PROGRAM MAIN
VAR
    rTrig : R_TRIG;
END_VAR

rTrig(CLK := GVL.BoutonSelecteur);

GVL.LumiereDroite := FALSE;
GVL.LumiereGauche := FALSE;

IF GVL.BoutonVirtuel THEN
    IF GVL.BoutonSelecteur THEN
        GVL.LumiereDroite := TRUE;
    ELSE
        GVL.LumiereGauche := TRUE;
    END_IF
END_IF;

IF rTrig.Q AND GVL.BoutonVirtuel THEN
    IF GVL.BoutonSelecteur THEN
        GVL.CounterLumiereDroiteAllumer := GVL.CounterLumiereDroiteAllumer + 1;
    ELSE
        GVL.CounterLumiereGaucheAllumer := GVL.CounterLumiereGaucheAllumer + 1;
    END_IF
END_IF;

END_PROGRAM

(* stored: Version 1.1.0.1, ProductVersion 3.1.4024.16
   POU MAIN: Id {47fb85a4-8975-45bc-84a8-4e8406f2213d}, SpecialFunc None *)
